(*
SPDX-FileCopyrightText: © 2026 Oleksandr Tiutyk <trofimich@gmail.com>
SPDX-License-Identifier: MIT
License: https://opensource.org/license/mit
*)

(*!
<summary>
Beckhoff floating-point analog input channel process image.
</summary>
<description>
Encapsulates a 16-bit status word and a 32-bit single-precision REAL process value '%I*' for multi-range
analog input channels.
When used for I/O, link located fields or their containing buffers to the matching selected PDOs.
The record is not a packed wire buffer; compiler padding is not part of the device specification.
Unlinked/default values do not prove valid I/O. The caller evaluates bus/channel validity before use.
Use one owner task per instance and externally synchronize other access; multi-field snapshots are not atomic.
Copies store data without creating hardware links. Keep borrowed field references valid while consumers are bound.
This passive record performs no validation, synchronization, configuration or protocol advancement.
Select standard status-plus-value PDOs matching the declared Value type; compact value-only PDOs
are outside this model. Configure electrical range and scaling separately on the device.
</description>
*)
TYPE ANALOG_INPUT_REAL_CHANNEL :
STRUCT
	Status AT %I* : WORD;
	Value AT %I* : REAL;
END_STRUCT
END_TYPE

(* stored: Version 1.1.0.1, ProductVersion 3.1.4026.21
   DUT ANALOG_INPUT_REAL_CHANNEL: Id {4361d0c9-c2d1-4cff-b4d0-bc2e9ae63f5c} *)
